INTERFACE I_BinArg EXTENDS I_Arg

PROPERTY Val : LWORD
GET
END_GET
END_PROPERTY

END_INTERFACE

(* stored: Version 1.1.0.1
   Itf I_BinArg: Id {99093205-7065-4eb6-89a9-37c964f55e60}
   Property Val: Id {94f85ac0-4d08-4408-b0e5-fb1650d0d9ca}
   Get Get: Id {ebcefd7c-0c22-4573-ac8c-826e199e6bae} *)
